Staubli VAL3: CmdTxtReading.pgx

program CmdTxtReading()
begin
  call Txt_initData()
  call txt_PkgInit()
  ////  waitEndMove()
  nCycleTotal=200
  while true
    //if n_sTxt<nTxtTotal and nTxtTotal>2
    if n_Roate<nCycleTotal and nTxtTotal>2
      if bTxt1==true
        call TxtReadRoom1()
      else
      endIf
      if bTxt2==true
        call TxtReadRoom2()
      else
      endIf
      if bTxt3==true
        call TxtReadRoom3()
      else
      endIf
    else
    endIf
    //    nScrPts=n_sTxt
    //    call hmi_refreshmain()
    delay(0)
  endWhile
end
